(*
  QualiVision line camera system
  DMAX76.   
*)
FUNCTION_BLOCK FB_LineCamera76 EXTENDS FB_LineCamera

VAR CONSTANT
  cCameraWidth76            : DINT :=  9216;   (*Camera width [px]*)
  cCameraMechOffsetTC76     : REAL := 101.5;   (*Camera mechanical offset at calibration temp [mm]*)
  cMechOffsetCameraToPU76   : REAL :=  13.039; (*Camera mechanical offset to PrintUnit [mm]*)
  cPrintUnitMechOffsetTC76  : REAL := 32.9869; (*PrintUnit mechanical offset at calibration temp [mm]*)
END_VAR

SUPER^();

METHOD InitLineCamera
VAR_INPUT
  nPrintUnitResolution         : UDINT;    (*printhead pixel resolution [dpi]*)
  nPrintUnitSubPx              : UDINT;    (*print unit subPixel resolution [SubPx]*)
  nPrintUnitWidth              : UDINT;    (*print unit width in [px]*)
  iCameraTrigger               : I_CameraTrigger;
END_VAR
(*Init for dmax type*)
_nCameraWidth           := cCameraWidth76;
_fCameraMechOffsetTC    := cCameraMechOffsetTC76;
_fMechOffsetCameraToPU  := cMechOffsetCameraToPU76;
_fPrintUnitMechOffsetTC := cPrintUnitMechOffsetTC76;

SUPER^.InitLineCamera( nPrintUnitResolution := nPrintUnitResolution
                      , nPrintUnitSubPx := nPrintUnitSubPx
                      , nPrintUnitWidth := nPrintUnitWidth
                      , iCameraTrigger := iCameraTrigger);
END_METHOD

{attribute 'monitoring':='variable'}
PROPERTY sName : STRING
GET
sName := 'LineCam 76';
END_GET
END_PROPERTY

END_FUNCTION_BLOCK

(* stored: Version 1.1.0.1, ProductVersion 3.1.4024.3
   POU FB_LineCamera76: Id {f026dcfb-030e-4811-bbfc-3ae7c59e9f6d}, SpecialFunc None
   Method InitLineCamera: Id {1ec7c9de-71b9-42c5-a620-6c5cf1b0cd9c}
   Property sName: Id {8415e38e-99a3-4cdd-944c-e2e705dec557}
   Get Get: Id {bbd80cc0-17e9-4b46-add2-0076879e7d29} *)
